TYPE DUT :
STRUCT
END_STRUCT
END_TYPE

(* stored: Version 1.1.0.1, ProductVersion 3.1.4024.12
   DUT DUT: Id {c9ea8f26-32d4-439f-b929-3a4241c85c69} *)
